(*
SPDX-FileCopyrightText: © 2026 Oleksandr Tiutyk <trofimich@gmail.com>
SPDX-License-Identifier: MIT
License: https://opensource.org/license/mit
*)

(*!
<summary>Stores a sequence of bytes with fixed or dynamic capacity.</summary>
<description>
CreateEnumerator allocates an independent cursor owned by its caller. The collection must remain alive while
that cursor is used. Static capacity zero selects dynamic storage; otherwise bytes reside in the instance.
DataAddress exposes internal storage: external reassignment invalidates the collection, and growth or
Clear(TRUE) invalidates borrowed addresses. Raw copy methods do not adopt input memory. Remove by value leaves
the collection unchanged when no match exists, including on an empty dynamic instance. WriteData centralizes
capacity checks, writes and buffer replacement. Internal sources and overlapping ranges are supported when the
full source range is readable; growth keeps the old buffer alive until copying completes. Derived callers of
WriteData must satisfy its validated-input preconditions.
Instances cannot be assigned by value: copying backing pointers or disposal responsibility would create
unsafe aliases. Interface references still borrow this instance; copying an interface does not clone storage.
</description>
*)

{attribute 'no_explicit_call' := 'do not call this function block directly'}
FUNCTION_BLOCK ByteList 
VAR_GENERIC CONSTANT
	{attribute 'hide'} 
	//! <summary>Inline capacity; zero selects dynamic backing storage.</summary>
	_StaticCapacity : TOF_Core.DINT_LENGTH := 0;
END_VAR
EXTENDS TOF_Core.Object IMPLEMENTS IByteList
VAR_OUTPUT
	//! <summary>Borrows backing bytes; growth or released capacity invalidates the address.</summary>
	DataAddress : POINTER TO BYTE;
END_VAR
VAR_STAT
	//! <summary>Class name shared by all instances of this function block.</summary>
	{attribute 'hide'} 
	_ClassName : STRING := __POUNAME();
END_VAR
VAR
	{attribute 'hide'} 
	_StaticArray : ARRAY [0.._StaticCapacity - 1] OF BYTE;
	
	{attribute 'hide'} 
	_DynamicCapacity : TOF_Core.DINT_LENGTH;
	{attribute 'hide'} 
	_Length : DINT;
END_VAR

(*!
<summary>Appends the raw storage bytes of an ANY argument.</summary>
<description>
Borrows the argument for copying and uses its full runtime size, including string capacity and structure
padding. Not portable serialization or object cloning. Shares AppendData capacity checks, overlap support and
failure behavior. Descendants cannot override this storage operation; capacity, indexing and disposal remain
governed by this collection implementation.
</description>
*)
METHOD FINAL AppendAny : IByteList
VAR_INPUT
	data : ANY;
END_VAR
AppendAny := AppendData(data := data.pValue, dataSize := TO_DINT(data.diSize));
END_METHOD

(*!
<summary>Appends one byte by value.</summary>
<description>
Returns this list. Full static storage raises an exception; dynamic growth uses checked allocation and
terminal OOM handling. Descendants cannot override this storage operation; capacity, indexing and disposal
remain governed by this collection implementation.
</description>
*)
METHOD FINAL AppendByte : IByteList
VAR_INPUT
	value : BYTE;
END_VAR
AppendByte := AppendData(data := ADR(value), dataSize := 1);
END_METHOD

(*!
<summary>Appends bytes copied from a borrowed memory range.</summary>
<description>
Null data or zero dataSize is a no-op before size validation. Otherwise the source must be readable and
negative sizes or a resulting length outside DINT raise ArgumentOutOfRangeException before copying. Static
capacity exhaustion raises StaticCollectionFullException. Dynamic allocation uses checked growth and terminal
OOM handling. The existing growth increment (free capacity plus input size) is retained and must also fit. The
source may refer to this collection buffer, including overlapping ranges. The caller must provide a readable
range of dataSize bytes; growth keeps the old buffer alive until copying completes. No restriction to logical
Length is imposed on the source. Returns this list. Descendants cannot override this storage operation;
capacity, indexing and disposal remain governed by this collection implementation.
</description>
*)
METHOD FINAL AppendData : IByteList
VAR_INPUT
	data : POINTER TO BYTE;
	dataSize : TOF_Core.DINT_LENGTH;
END_VAR
AppendData := THIS^;

IF data = 0 OR_ELSE dataSize = TOF_Core.SignedInt32.ZERO THEN
	RETURN;
END_IF

IF dataSize < TOF_Core.SignedInt32.ZERO
	OR_ELSE dataSize > TOF_Core.SignedInt32.MAX_VALUE - _Length
THEN
	TOF_Core.Exceptions.ThrowArgumentOutOfRange(
		sourceNamespaceName := NamespaceName,
		sourceClassName := ClassName,
		sourcePOUName := __POUNAME(),
		sourcePosition := __POSITION(),
		argumentName := 'dataSize',
		argumentValue := dataSize
	);
END_IF

WriteData(
	data := data,
	dataSize := dataSize,
	startIndex := _Length,
	requestedCapacity := TO_ULINT(Capacity) + TO_ULINT(Capacity - _Length) + TO_ULINT(dataSize)
);
END_METHOD

(*!
<summary>Appends the raw bytes referenced by a generic descriptor.</summary>
<description>
Borrows the descriptor without adopting or releasing it. Copies Address and Size without value conversion or
object cloning. Size above SignedInt32.MAX_VALUE raises ArgumentOutOfRangeException before narrowing,
including for a null Address. Shares AppendData aliasing and failure behavior. Descendants cannot override
this storage operation; capacity, indexing and disposal remain governed by this collection implementation.
</description>
*)
METHOD FINAL AppendGeneric : IByteList
VAR_INPUT
	data : TOF_Core.GENERIC_VALUE;
END_VAR
IF data.Size > TO_ULINT(TOF_Core.SignedInt32.MAX_VALUE) THEN
	TOF_Core.Exceptions.ThrowArgumentOutOfRange(
		sourceNamespaceName := NamespaceName,
		sourceClassName := ClassName,
		sourcePOUName := __POUNAME(),
		sourcePosition := __POSITION(),
		argumentName := 'data.Size',
		argumentValue := data.Size
	);
END_IF

AppendGeneric := AppendData(data := data.Address, dataSize := TO_DINT(data.Size));
END_METHOD

(*!
<summary>Reports the currently allocated number of slots.</summary>
<description>
Units are bytes for ByteList and entries for other collections. Static capacity is fixed; dynamic capacity can
change on growth or clearing. This is not a guarantee that the next allocation succeeds.
</description>
*)
{attribute 'monitoring' := 'call'}
PROPERTY FINAL Capacity : TOF_Core.DINT_LENGTH
GET
Capacity := SEL(_StaticCapacity = 0, _StaticCapacity, _DynamicCapacity);
END_GET
END_PROPERTY

(*!
<summary>Borrows the concrete collection class name without transferring storage ownership.</summary>
*)
{attribute 'monitoring' := 'call'}
PROPERTY ClassName : REFERENCE TO STRING
GET
ClassName REF= _ClassName;
END_GET
END_PROPERTY

(*!
<summary>Resets the byte count and optionally releases dynamic storage.</summary>
<description>
The default retains capacity for reuse. releaseDynamicMemory = TRUE deletes dynamic storage and sets capacity
to zero. Static storage is retained. Returns this list; old contents are no longer logical entries.
Descendants cannot override this storage operation; capacity, indexing and disposal remain governed by this
collection implementation.
</description>
*)
METHOD FINAL Clear : IByteList
VAR_INPUT
	releaseDynamicMemory : BOOL := FALSE;
END_VAR
Clear := THIS^;

IF releaseDynamicMemory AND_THEN Dynamic AND_THEN _DynamicCapacity > 0 THEN
	__DELETE(DataAddress);
	_DynamicCapacity := 0;
END_IF

_Length := 0;
END_METHOD

(*!
<summary>Creates an independent enumerator owned by the caller.</summary>
<description>
The caller must explicitly release the enumerator and keep this collection alive while using it. Allocation
failure invokes DynamicMemoryManager.RaiseAllocationFailure without a heap exception; it is terminal and is
not returned as a recoverable null result.
</description>
*)
METHOD CreateEnumerator : TOF_Core.IEnumerator
VAR
	enumerator : POINTER TO ByteListEnumerator;
END_VAR
enumerator := __NEW(ByteListEnumerator(list := THIS^));

IF enumerator = 0 THEN
	TOF_Core.DynamicMemoryManager.RaiseAllocationFailure();
END_IF

CreateEnumerator := enumerator^;
END_METHOD

(*!
<summary>Reports whether storage can grow dynamically.</summary>
<description>
Static capacity zero selects dynamic storage. Dynamic collections can still fail to allocate.
</description>
*)
{attribute 'monitoring' := 'call'}
PROPERTY FINAL Dynamic : BOOL
GET
Dynamic := _StaticCapacity = 0;
END_GET
END_PROPERTY

(*!
<summary>Reports whether the collection has no entries.</summary>
<description>
Reflects Length; not a check of payload lifetime or memory health.
</description>
*)
{attribute 'monitoring' := 'call'}
PROPERTY FINAL Empty : BOOL
GET
Empty := _Length <= 0;
END_GET
END_PROPERTY

(*!
<summary>Releases dynamic byte storage during destruction.</summary>
<description>
Calls Clear(releaseDynamicMemory := TRUE); inline storage is not separately deleted. Lifecycle methods must complete without
exceptions. No separate copy-code ownership handoff is implemented.
</description>
*)

METHOD FB_exit : BOOL
VAR_INPUT
	bInCopyCode : BOOL; 
END_VAR
Clear(releaseDynamicMemory := TRUE);
END_METHOD

(*!
<summary>Binds inline byte storage for a static instance.</summary>
<description>
No allocation or callbacks are performed. Dynamic instances start without a backing buffer. No explicit
online-change relocation repair is implemented.
</description>
*)
METHOD FB_init : BOOL
VAR_INPUT
	bInitRetains : BOOL; // TRUE: the retain variables are initialized (reset warm / reset cold)
	bInCopyCode : BOOL; // TRUE: the instance will be copied to the copy code afterward (online change)
END_VAR
IF NOT Dynamic THEN
	DataAddress := ADR(_StaticArray); 
END_IF
END_METHOD

(*!
<summary>Finds the first occurrence of a byte.</summary>
<description>
Searches from zero. TRUE makes index valid; on FALSE no index is promised. The collection is unchanged.
Descendants cannot override this storage operation; capacity, indexing and disposal remain governed by this
collection implementation.
</description>
*)
METHOD FINAL Find : BOOL
VAR_INPUT
	value : BYTE;
END_VAR
VAR_OUTPUT
	index : TOF_Core.DINT_INDEX;
END_VAR
VAR
	i : DINT;	
END_VAR
IF _Length > 0 THEN
	FOR i := 0 TO _Length - 1 DO
		IF DataAddress[i] = value THEN
			index := i;
			Find := TRUE;
			RETURN;
		END_IF 	
	END_FOR
END_IF
END_METHOD

(*!
<summary>Reports whether fixed-capacity storage has no free slot.</summary>
<description>
Dynamic collections report FALSE even when Length equals Capacity. This does not guarantee available heap
memory.
</description>
*)
{attribute 'monitoring' := 'call'}
PROPERTY FINAL Full : BOOL
GET
Full := _StaticCapacity <> 0 AND_THEN _Length >= _StaticCapacity;
END_GET
END_PROPERTY

(*!
<summary>Returns the byte at an existing zero-based position.</summary>
<description>
Raises an exception when backing storage is absent or the index is outside Length. The result is a byte copy.
Descendants cannot override this storage operation; capacity, indexing and disposal remain governed by this
collection implementation.
</description>
*)
METHOD FINAL Get : BYTE
VAR_INPUT
	index : TOF_Core.DINT_INDEX;
END_VAR
IF DataAddress = 0 THEN
	TOF_Core.Exceptions.ThrowStandard(
		sourceNamespaceName := NamespaceName,
		sourceClassName := ClassName,
		sourcePOUName := __POUNAME(),
		sourcePosition := __POSITION(),
		message := "Dynamic byte array is empty"
	);
END_IF

IF index < 0 THEN
	TOF_Core.Exceptions.ThrowStandard(
		sourceNamespaceName := NamespaceName,
		sourceClassName := ClassName,
		sourcePOUName := __POUNAME(),
		sourcePosition := __POSITION(),
		message := "Index is less then zero"
	);
END_IF

IF index >= _Length THEN
	TOF_Core.Exceptions.ThrowStandard(
		sourceNamespaceName := NamespaceName,
		sourceClassName := ClassName,
		sourcePOUName := __POUNAME(),
		sourcePosition := __POSITION(),
		message := "Index is too large"
	);
END_IF

Get := DataAddress[index];
END_METHOD

(*!
<summary>Reports the number of stored entries.</summary>
<description>
Units are bytes for ByteList and entries for other collections. Existing positions range from zero through
Length minus one.
</description>
*)
{attribute 'monitoring' := 'call'}
PROPERTY FINAL Length : TOF_Core.DINT_LENGTH
GET
Length := _Length;
END_GET
END_PROPERTY

(*!
<summary>Loads the full raw representation of an ANY argument at a position.</summary>
<description>
Delegates to LoadFromData using the runtime byte size, including padding and string capacity. Borrows the
source and may truncate the previous tail. Shares LoadFromData limits; not portable serialization. Descendants
cannot override this storage operation; capacity, indexing and disposal remain governed by this collection
implementation.
</description>
*)
METHOD FINAL LoadFromAny : IByteList
VAR_INPUT
	data : ANY;
	startIndex : TOF_Core.DINT_INDEX := 0;
END_VAR
LoadFromAny := LoadFromData(data := data.pValue, dataSize := TO_DINT(data.diSize), startIndex := startIndex);
END_METHOD

(*!
<summary>Copies bytes at a position and sets Length to the end of the copy.</summary>
<description>
startIndex must lie between zero and old Length inclusive, and dataSize must be nonnegative; invalid arguments
raise ArgumentOutOfRangeException. Null data or zero size leaves Length unchanged after these checks. For a
nonempty copy, the resulting length is checked against DINT before arithmetic or mutation. The prefix remains
and the tail beyond the new end is logically truncated. Static capacity exhaustion raises
StaticCollectionFullException; dynamic growth uses checked allocation and terminal OOM handling. Internal
sources and overlapping ranges are supported. The caller must provide a readable source range of dataSize
bytes; the old buffer remains alive throughout copying on growth. No restriction to logical Length is imposed
on the source. Returns this list. Descendants cannot override this storage operation; capacity, indexing and
disposal remain governed by this collection implementation.
</description>
*)
METHOD FINAL LoadFromData : IByteList
VAR_INPUT
	data : POINTER TO BYTE;
	dataSize : TOF_Core.DINT_LENGTH;
	startIndex : TOF_Core.DINT_INDEX := 0;
END_VAR
IF startIndex < TOF_Core.SignedInt32.ZERO OR_ELSE startIndex > _Length THEN
	TOF_Core.Exceptions.ThrowArgumentOutOfRange(
		sourceNamespaceName := NamespaceName,
		sourceClassName := ClassName,
		sourcePOUName := __POUNAME(),
		sourcePosition := __POSITION(),
		argumentName := 'startIndex',
		argumentValue := startIndex
	);
END_IF

IF dataSize < TOF_Core.SignedInt32.ZERO THEN
	TOF_Core.Exceptions.ThrowArgumentOutOfRange(
		sourceNamespaceName := NamespaceName,
		sourceClassName := ClassName,
		sourcePOUName := __POUNAME(),
		sourcePosition := __POSITION(),
		argumentName := 'dataSize',
		argumentValue := dataSize
	);
END_IF

LoadFromData := THIS^;
 
IF data = 0 OR_ELSE dataSize = TOF_Core.SignedInt32.ZERO THEN
	RETURN;
END_IF

IF dataSize > TOF_Core.SignedInt32.MAX_VALUE - startIndex THEN
	TOF_Core.Exceptions.ThrowArgumentOutOfRange(
		sourceNamespaceName := NamespaceName,
		sourceClassName := ClassName,
		sourcePOUName := __POUNAME(),
		sourcePosition := __POSITION(),
		argumentName := 'dataSize',
		argumentValue := dataSize
	);
END_IF

WriteData(
		data := data,
		dataSize := dataSize,
		startIndex := startIndex,
		requestedCapacity := TO_ULINT(startIndex) + TO_ULINT(dataSize)
	);
END_METHOD

(*!
<summary>Loads the byte range referenced by a generic descriptor.</summary>
<description>
Borrows the descriptor without adoption or release. Size above SignedInt32.MAX_VALUE raises
ArgumentOutOfRangeException before narrowing, including for a null Address. Shares LoadFromData index checks,
truncation, aliasing and failure behavior. Descendants cannot override this storage operation; capacity,
indexing and disposal remain governed by this collection implementation.
</description>
*)
METHOD FINAL LoadFromGeneric : IByteList
VAR_INPUT
	data : TOF_Core.GENERIC_VALUE;
	startIndex : TOF_Core.DINT_INDEX := 0;
END_VAR
IF data.Size > TO_ULINT(TOF_Core.SignedInt32.MAX_VALUE) THEN
	TOF_Core.Exceptions.ThrowArgumentOutOfRange(
		sourceNamespaceName := NamespaceName,
		sourceClassName := ClassName,
		sourcePOUName := __POUNAME(),
		sourcePosition := __POSITION(),
		argumentName := 'data.Size',
		argumentValue := data.Size
	);
END_IF

LoadFromGeneric := LoadFromData(data := data.Address, dataSize := TO_DINT(data.Size), startIndex := startIndex);
END_METHOD

(*!
<summary>Provides the library namespace for diagnostics.</summary>
<description>
Borrowed read-only reference to compiler-initialized metadata; no ownership transfer.
</description>
*)
{attribute 'monitoring' := 'call'}
PROPERTY NamespaceName : REFERENCE TO STRING
GET
NamespaceName REF= CurrentNamespace.Name;
END_GET
END_PROPERTY

(*!
<summary>Removes the first occurrence of a byte if present.</summary>
<description>
Removes only the first matching byte, compacts later bytes through RemoveAt and returns this list. An absent
value or an empty static or dynamic list leaves the collection unchanged without raising an exception for
absence. Capacity is retained. Requires an intact collection whose backing storage remains valid for its
logical contents. Descendants cannot override this storage operation; capacity, indexing and disposal remain
governed by this collection implementation.
</description>
*)
METHOD FINAL Remove : IByteList
VAR_INPUT
	value : BYTE;
END_VAR
VAR
	index : DINT;
END_VAR
Remove := THIS^;

IF Find(value := value, index => index) THEN
	RemoveAt(index := index, count := 1);
END_IF
END_METHOD

(*!
<summary>Removes a contiguous byte range and compacts remaining bytes.</summary>
<description>
Requires an existing index and a nonnegative count no greater than the remaining length; otherwise raises
ArgumentOutOfRangeException. The range is checked by subtraction before computing its end. Zero count is a
no-op only after index validation. Capacity is retained. Returns this list. Descendants cannot override this
storage operation; capacity, indexing and disposal remain governed by this collection implementation.
</description>
*)
METHOD FINAL RemoveAt : IByteList
VAR_INPUT
	index : TOF_Core.DINT_INDEX;
	count : TOF_Core.DINT_LENGTH := 1;
END_VAR
IF index < TOF_Core.SignedInt32.ZERO OR_ELSE index >= _Length THEN
	TOF_Core.Exceptions.ThrowArgumentOutOfRange(
		sourceNamespaceName := NamespaceName,
		sourceClassName := ClassName,
		sourcePOUName := __POUNAME(),
		sourcePosition := __POSITION(),
		argumentName := 'index',
		argumentValue := index
	);
END_IF

IF count < TOF_Core.SignedInt32.ZERO OR_ELSE count > _Length - index THEN
	TOF_Core.Exceptions.ThrowArgumentOutOfRange(
		sourceNamespaceName := NamespaceName,
		sourceClassName := ClassName,
		sourcePOUName := __POUNAME(),
		sourcePosition := __POSITION(),
		argumentName := 'count',
		argumentValue := count
	);
END_IF

RemoveAt := THIS^;

IF count = TOF_Core.SignedInt32.ZERO THEN
	RETURN;
END_IF

IF count <> _Length THEN
	Tc2_System.MEMMOVE(
		destAddr := DataAddress + TO_LWORD(index),
		srcAddr := DataAddress + TO_LWORD(index + count),
		n := TO_UDINT(_Length - index - count)
	);
END_IF

_Length := _Length - count;
END_METHOD

(*!
<summary>Reports the size of this function-block instance.</summary>
<description>
Measured in bytes; includes inline storage but excludes separately allocated buffers, payload and enumerators.
</description>
*)
{attribute 'monitoring' := 'call'}
PROPERTY SelfSize : ULINT
GET
SelfSize := XSIZEOF(THIS^);
END_GET
END_PROPERTY

(*!
<summary>Overwrites one existing byte.</summary>
<description>
Requires allocated storage and an index within Length; otherwise raises an exception. Length and Capacity are
unchanged. Returns this list. Descendants cannot override this storage operation; capacity, indexing and
disposal remain governed by this collection implementation.
</description>
*)
METHOD FINAL Set : IByteList
VAR_INPUT
	index : TOF_Core.DINT_INDEX;
	value : BYTE;
END_VAR
IF DataAddress = 0 THEN
	TOF_Core.Exceptions.ThrowStandard(
		sourceNamespaceName := NamespaceName,
		sourceClassName := ClassName,
		sourcePOUName := __POUNAME(),
		sourcePosition := __POSITION(),
		message := "Dynamic byte array is empty"
	);
END_IF

IF index < 0 THEN
	TOF_Core.Exceptions.ThrowStandard(
		sourceNamespaceName := NamespaceName,
		sourceClassName := ClassName,
		sourcePOUName := __POUNAME(),
		sourcePosition := __POSITION(),
		message := "Index is less then zero"
	);
END_IF

IF index >= _Length THEN
	TOF_Core.Exceptions.ThrowStandard(
		sourceNamespaceName := NamespaceName,
		sourceClassName := ClassName,
		sourcePOUName := __POUNAME(),
		sourcePosition := __POSITION(),
		message := "Index is too large"
	);
END_IF

Set := THIS^;

DataAddress[index] := value;
END_METHOD

(*!
<summary>Writes a prepared byte range and centrally manages any buffer replacement.</summary>
<description>
The caller must validate a non-null readable source, positive dataSize, startIndex within Length and a
representable resulting length. requestedCapacity specifies the growth policy and is used only when the write
exceeds Capacity. It must cover the resulting length and fit DINT. Static exhaustion raises
StaticCollectionFullException. Invalid growth capacity raises ArgumentOutOfRangeException. Null NEW invokes
terminal allocation failure before mutation. Without growth, MEMMOVE supports overlapping ranges. With growth,
the old buffer remains alive until both existing bytes and source bytes have been copied; only then are
pointer, capacity and length committed and the old allocation deleted. Source ranges may include the
collection buffer, provided the full range is readable; no restriction to logical Length is imposed. Borrowed
buffer addresses are invalidated by growth. This helper does not validate arbitrary pointer lifetime.
</description>
*)
METHOD PROTECTED FINAL WriteData
VAR_INPUT
	data : POINTER TO BYTE;
	dataSize : TOF_Core.DINT_LENGTH;
	startIndex : TOF_Core.DINT_INDEX;
	requestedCapacity : ULINT;
END_VAR
VAR
	newLength : DINT;
	newMemory : POINTER TO BYTE;
	oldMemory : POINTER TO BYTE;

END_VAR
newLength := startIndex + dataSize;

IF newLength <= Capacity THEN
	Tc2_System.MEMMOVE(destAddr := DataAddress + TO_DWORD(startIndex), srcAddr := data, n := TO_UDINT(dataSize));
	_Length := newLength;
	RETURN;
END_IF

IF NOT Dynamic THEN
	TOF_Core.Exceptions.ThrowStaticCollectionFull(
		sourceNamespaceName := NamespaceName,
		sourceClassName := ClassName,
		sourcePOUName := __POUNAME(),
		sourcePosition := __POSITION(),
		collectionName := GetName(),
		capacity := TO_UDINT(Capacity)
	);
END_IF

IF requestedCapacity < TO_ULINT(newLength)
	OR_ELSE requestedCapacity > TO_ULINT(TOF_Core.SignedInt32.MAX_VALUE)
THEN
	TOF_Core.Exceptions.ThrowArgumentOutOfRange(
		sourceNamespaceName := NamespaceName,
		sourceClassName := ClassName,
		sourcePOUName := __POUNAME(),
		sourcePosition := __POSITION(),
		argumentName := 'capacity',
		argumentValue := requestedCapacity
	);
END_IF

newMemory := __NEW(BYTE, TO_UDINT(requestedCapacity));

IF newMemory = 0 THEN
	TOF_Core.DynamicMemoryManager.RaiseAllocationFailure();
END_IF

oldMemory := DataAddress;

IF _Length > TOF_Core.SignedInt32.ZERO THEN
	Tc2_System.MEMCPY(destAddr := newMemory, srcAddr := oldMemory, n := TO_UDINT(_Length));
END_IF

// The source may refer to the old buffer, which remains alive until this copy completes.
Tc2_System.MEMCPY(destAddr := newMemory + TO_DWORD(startIndex), srcAddr := data, n := TO_UDINT(dataSize));

DataAddress := newMemory;
_DynamicCapacity := TO_DINT(requestedCapacity);
_Length := newLength;

IF oldMemory <> 0 THEN
	__DELETE(oldMemory);
END_IF
END_METHOD

END_FUNCTION_BLOCK

(* stored: Version 1.1.0.1
   POU ByteList: Id {44085af7-7241-03f1-3e6d-aeb87f0c58dd}, SpecialFunc None
   Folder Service methods: Id {685c0c64-63d7-45b0-8d80-202fe70951c4}
   Method AppendAny: Id {fa939ac2-b614-4bc3-8ef3-f524865ffb5f}
   Method AppendByte: Id {90a35576-aaee-0fbc-214a-d1c0f81c72fb}
   Method AppendData: Id {d35c3ee4-7daa-49d5-be43-e476b3efb046}
   Method AppendGeneric: Id {ac72fb80-d130-4ae7-81e5-86ab3708db48}
   Property Capacity: Id {3ae8e9be-a7d0-403a-8d29-c44983ebf381}
   Get Get: Id {b809a1de-e3ae-4897-8390-093667992014}
   Property ClassName: Id {3b9bf934-b83c-0948-370d-5e8e28db661a}
   Get Get: Id {a74d6b23-00f3-0fef-283c-b96c5cad2f8b}
   Method Clear: Id {58795b0c-c9a9-0b7d-1801-4867f25906b7}
   Method CreateEnumerator: Id {9eb1bbc5-e145-4b1d-be02-fc14e3a7b7c4}
   Property Dynamic: Id {7fc86655-965e-4584-8395-7f580dc2445d}
   Get Get: Id {8c679524-cf9f-40aa-9def-10c089c4abae}
   Property Empty: Id {8cac260d-f211-4946-9f91-204b369e9bc6}
   Get Get: Id {cdc3f172-a10e-45a6-be1f-94a4244848e7}
   Method FB_exit: Id {58cee31c-ede5-0b41-17b5-f6dfb8c1dea7}
   Method FB_init: Id {9b89d2ed-7216-4482-ba21-51df798725b2}
   Method Find: Id {f870e801-4961-0438-0486-eeff60dc3fea}
   Property Full: Id {fb559251-67ca-4284-974d-f6b046168be3}
   Get Get: Id {a258343f-e2ac-4ae3-91ec-9e66c42b2a82}
   Method Get: Id {7a2d32dc-2bf1-07fe-3b69-aed2ad5b300d}
   Property Length: Id {d1b0052d-4e1b-09cb-235e-e87df6b9b5a5}
   Get Get: Id {457f3f94-ecd5-03a2-1012-5eb779d04c66}
   Method LoadFromAny: Id {6ca12394-c5fc-0274-1ee4-d0bfc0727c06}
   Method LoadFromData: Id {9fe65b5e-87b5-0537-23bd-6a15d825d74e}
   Method LoadFromGeneric: Id {803d0535-a6e1-4d89-878a-9e90b4d80911}
   Property NamespaceName: Id {6affa192-b708-4407-b07b-3f99b221293a}
   Get Get: Id {08e774db-64ad-4b08-8c9f-7cf3351a9ee4}
   Method Remove: Id {bf82b30e-92dd-0d23-0038-cce05024df18}
   Method RemoveAt: Id {13c7901e-f730-033f-2407-dd64a3fc2480}
   Property SelfSize: Id {eb116396-1c6b-495f-b284-5b142fa86f6c}
   Get Get: Id {9d568fff-ebc6-4d27-9dd9-94ca65277b07}
   Method Set: Id {7b62d34d-7ee9-07a4-2e13-b032abd0cd09}
   Method WriteData: Id {8ca653b8-50f7-445c-b10d-fbfed66a86d3} *)
